PROGRAM EtherCATComs //Handles all comunication over ethercat on ParamUpdate Task
VAR
	//QuickUpdate : FB_CheckIn_EtherCAT;
	ParamUpdate : FB_EtherCATReader;
	ParameterID_FromMom AT %I* : USINT;
	ParameterID_ToMom AT %Q*: USINT;
END_VAR

//ParamUpdate();
//ParameterID_ToMom := ParamUpdate.ID;
ParamUpdate();

END_PROGRAM

(* stored: Version 1.1.0.1, ProductVersion 3.1.4022.3
   POU EtherCATComs: Id {2abf7dcb-1891-4938-ad93-a08230d78e17}, SpecialFunc None *)
